TYPE TcoLiftingRotaryTransfer_Control EXTENDS TcoCore.TcoStruct:
STRUCT

	
		
END_STRUCT
END_TYPE

(* stored: Version 1.1.0.1
   DUT TcoLiftingRotaryTransfer_Control: Id {a6c11f95-7eb0-43d5-814f-9699bbf9148d} *)
